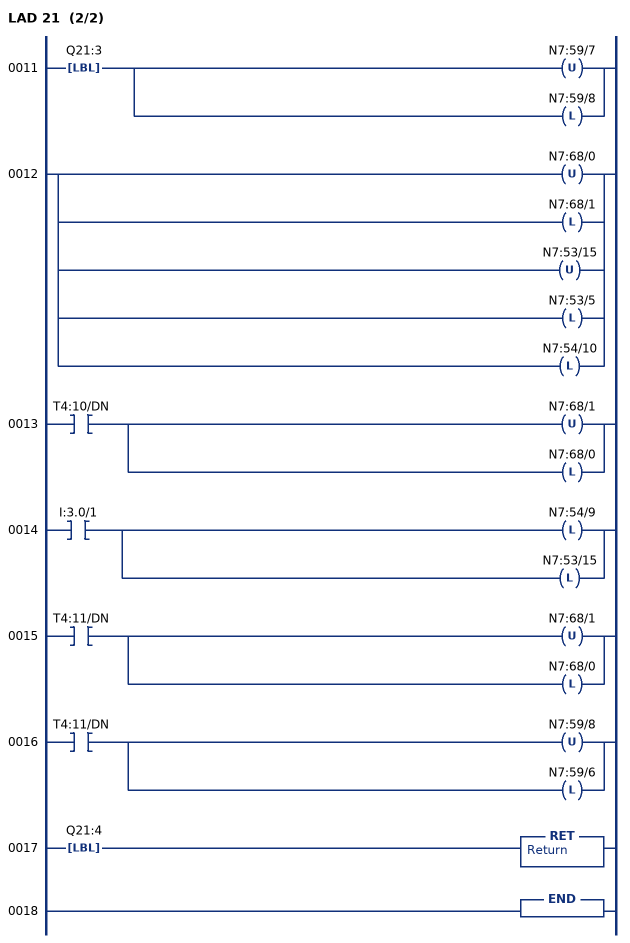
% Rung: 11 %
SOR LBL Q21:3 BST OTU N7:59/7 NXB OTL N7:59/8 BND EOR
% Rung: 12 %
SOR BST OTU N7:68/0 NXB OTL N7:68/1 NXB OTU N7:53/15 NXB OTL N7:53/5 NXB OTL N7:54/10 BND EOR
% Rung: 13 %
SOR XIC T4:10/DN BST OTU N7:68/1 NXB OTL N7:68/0 BND EOR
% Rung: 14 %
SOR XIC I:3.0/1 BST OTL N7:54/9 NXB OTL N7:53/15 BND EOR
% Rung: 15 %
SOR XIC T4:11/DN BST OTU N7:68/1 NXB OTL N7:68/0 BND EOR
% Rung: 16 %
SOR XIC T4:11/DN BST OTU N7:59/8 NXB OTL N7:59/6 BND EOR
% Rung: 17 %
SOR LBL Q21:4 RET EOR
% Rung: 18 %
SOR END EOR

LADDER 22
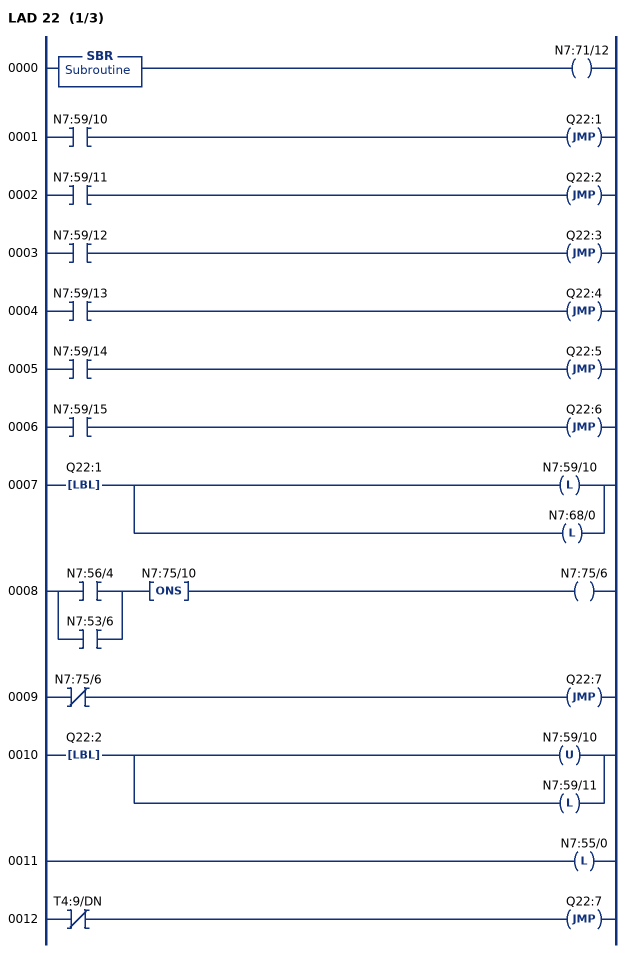
% Rung: 0 %
SOR SBR OTE N7:71/12 EOR
% Rung: 1 %
SOR XIC N7:59/10 JMP Q22:1 EOR
% Rung: 2 %
SOR XIC N7:59/11 JMP Q22:2 EOR
% Rung: 3 %
SOR XIC N7:59/12 JMP Q22:3 EOR
% Rung: 4 %
SOR XIC N7:59/13 JMP Q22:4 EOR
% Rung: 5 %
SOR XIC N7:59/14 JMP Q22:5 EOR
% Rung: 6 %
SOR XIC N7:59/15 JMP Q22:6 EOR
% Rung: 7 %
SOR LBL Q22:1 BST OTL N7:59/10 NXB OTL N7:68/0 BND EOR
% Rung: 8 %
SOR BST XIC N7:56/4 NXB XIC N7:53/6 BND OSR N7:75/10 OTE N7:75/6 EOR
% Rung: 9 %
SOR XIO N7:75/6 JMP Q22:7 EOR
% Rung: 10 %
SOR LBL Q22:2 BST OTU N7:59/10 NXB OTL N7:59/11 BND EOR
% Rung: 11 %
SOR OTL N7:55/0 EOR
% Rung: 12 %
SOR XIO T4:9/DN JMP Q22:7 EOR

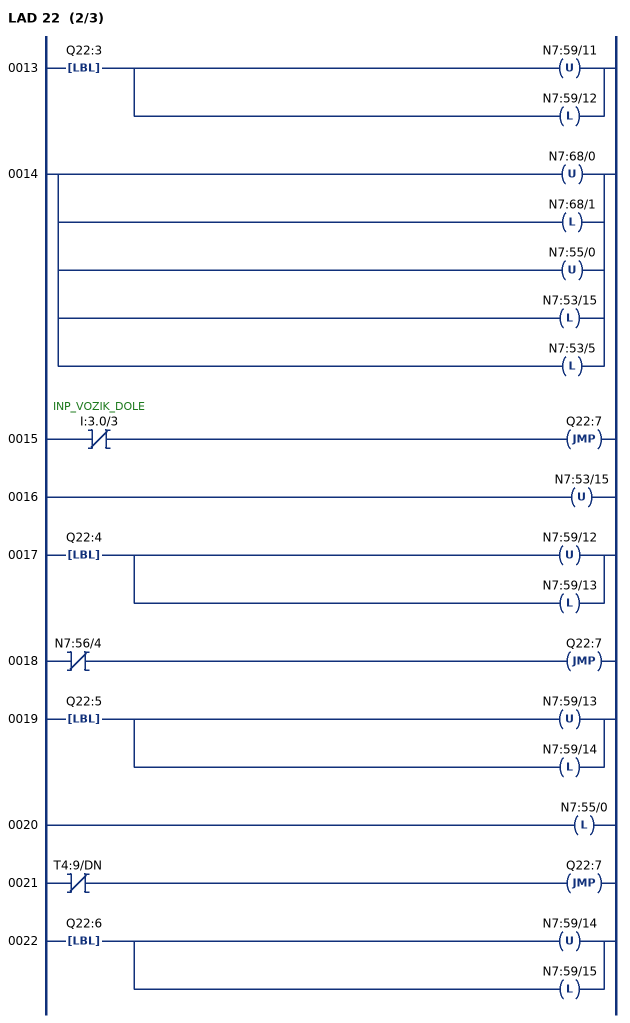
% Rung: 13 %
SOR LBL Q22:3 BST OTU N7:59/11 NXB OTL N7:59/12 BND EOR
% Rung: 14 %
SOR BST OTU N7:68/0 NXB OTL N7:68/1 NXB OTU N7:55/0 NXB OTL N7:53/15 NXB OTL N7:53/5 BND EOR
% Rung: 15 %
SOR XIO I:3.0/3 JMP Q22:7 EOR
%   I:3.0/3  INP_VOZIK_DOLE %
% Rung: 16 %
SOR OTU N7:53/15 EOR
% Rung: 17 %
SOR LBL Q22:4 BST OTU N7:59/12 NXB OTL N7:59/13 BND EOR
% Rung: 18 %
SOR XIO N7:56/4 JMP Q22:7 EOR
% Rung: 19 %
SOR LBL Q22:5 BST OTU N7:59/13 NXB OTL N7:59/14 BND EOR
% Rung: 20 %
SOR OTL N7:55/0 EOR
% Rung: 21 %
SOR XIO T4:9/DN JMP Q22:7 EOR
% Rung: 22 %
SOR LBL Q22:6 BST OTU N7:59/14 NXB OTL N7:59/15 BND EOR

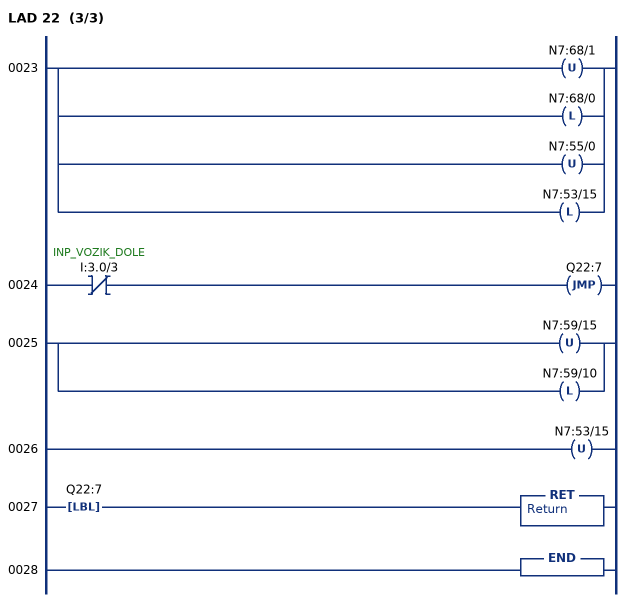
% Rung: 23 %
SOR BST OTU N7:68/1 NXB OTL N7:68/0 NXB OTU N7:55/0 NXB OTL N7:53/15 BND EOR
% Rung: 24 %
SOR XIO I:3.0/3 JMP Q22:7 EOR
%   I:3.0/3  INP_VOZIK_DOLE %
% Rung: 25 %
SOR BST OTU N7:59/15 NXB OTL N7:59/10 BND EOR
% Rung: 26 %
SOR OTU N7:53/15 EOR
% Rung: 27 %
SOR LBL Q22:7 RET EOR
% Rung: 28 %
SOR END EOR

LADDER 23
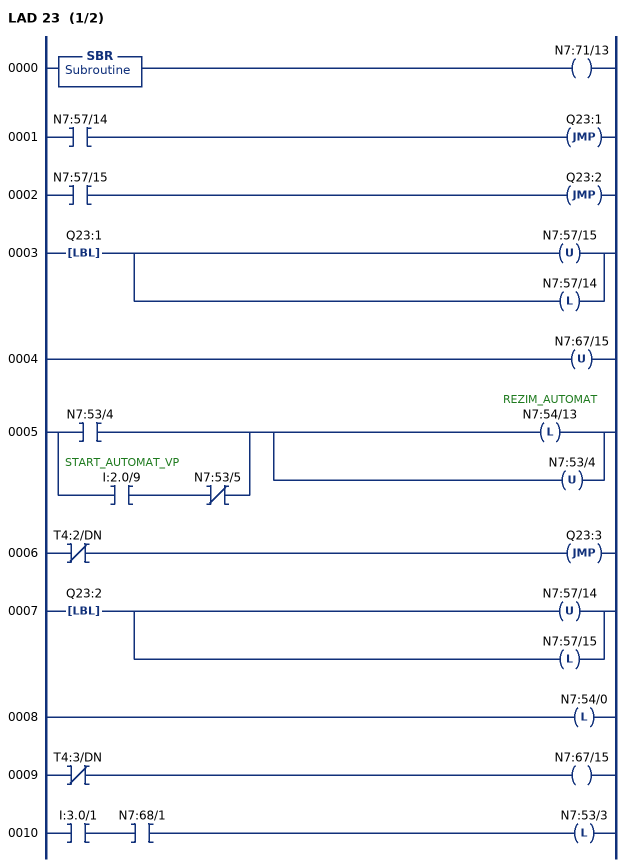
% Rung: 0 %
SOR SBR OTE N7:71/13 EOR
% Rung: 1 %
SOR XIC N7:57/14 JMP Q23:1 EOR
% Rung: 2 %
SOR XIC N7:57/15 JMP Q23:2 EOR
% Rung: 3 %
SOR LBL Q23:1 BST OTU N7:57/15 NXB OTL N7:57/14 BND EOR
% Rung: 4 %
SOR OTU N7:67/15 EOR
% Rung: 5 %
SOR BST XIC N7:53/4 NXB XIC I:2.0/9 XIO N7:53/5 BND BST OTL N7:54/13 NXB OTU N7:53/4 BND EOR
%   I:2.0/9  START_AUTOMAT_VP %
%   N7:54/13  REZIM_AUTOMAT %
% Rung: 6 %
SOR XIO T4:2/DN JMP Q23:3 EOR
% Rung: 7 %
SOR LBL Q23:2 BST OTU N7:57/14 NXB OTL N7:57/15 BND EOR
% Rung: 8 %
SOR OTL N7:54/0 EOR
% Rung: 9 %
SOR XIO T4:3/DN OTE N7:67/15 EOR
% Rung: 10 %
SOR XIC I:3.0/1 XIC N7:68/1 OTL N7:53/3 EOR

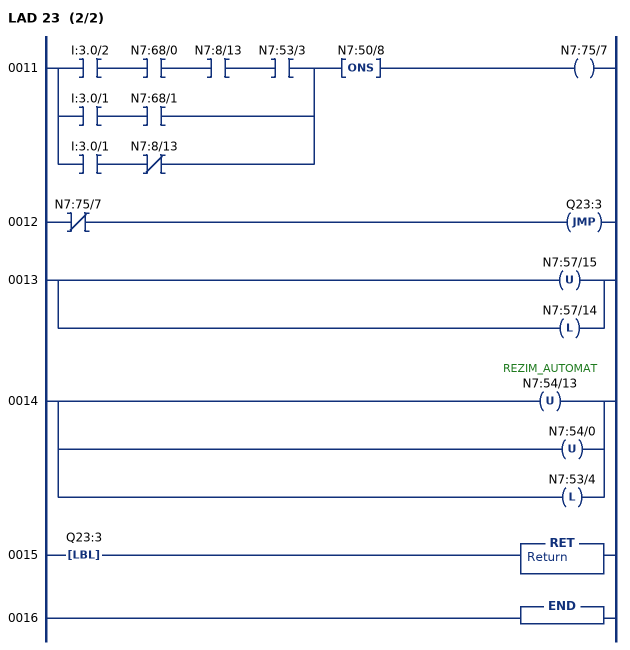
% Rung: 11 %
SOR BST XIC I:3.0/2 XIC N7:68/0 XIC N7:8/13 XIC N7:53/3 NXB XIC I:3.0/1 XIC N7:68/1 NXB XIC I:3.0/1 XIO N7:8/13 BND OSR N7:50/8 OTE N7:75/7 EOR
% Rung: 12 %
SOR XIO N7:75/7 JMP Q23:3 EOR
% Rung: 13 %
SOR BST OTU N7:57/15 NXB OTL N7:57/14 BND EOR
% Rung: 14 %
SOR BST OTU N7:54/13 NXB OTU N7:54/0 NXB OTL N7:53/4 BND EOR
%   N7:54/13  REZIM_AUTOMAT %
% Rung: 15 %
SOR LBL Q23:3 RET EOR
% Rung: 16 %
SOR END EOR

LADDER 24
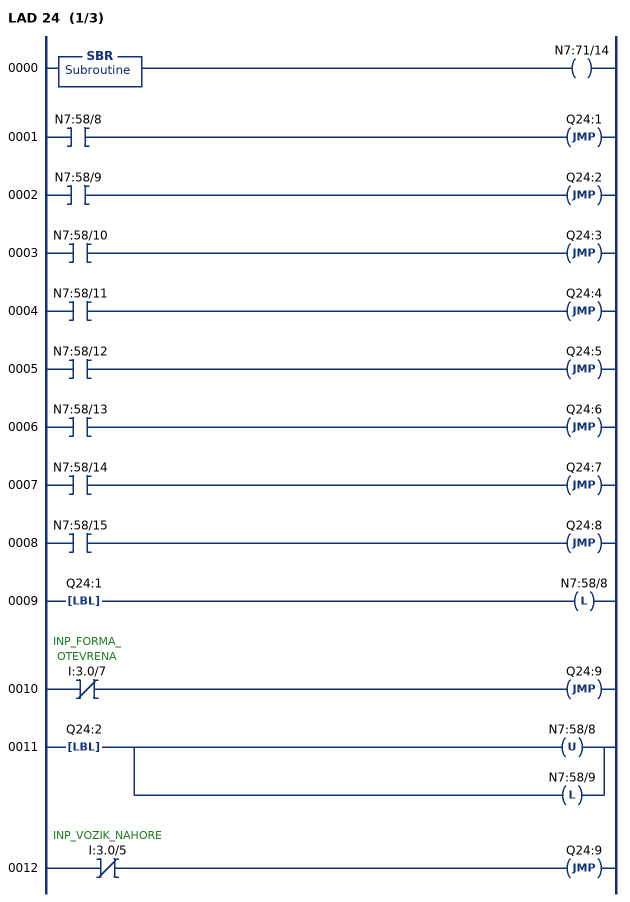
% Rung: 0 %
SOR SBR OTE N7:71/14 EOR
% Rung: 1 %
SOR XIC N7:58/8 JMP Q24:1 EOR
% Rung: 2 %
SOR XIC N7:58/9 JMP Q24:2 EOR
% Rung: 3 %
SOR XIC N7:58/10 JMP Q24:3 EOR
% Rung: 4 %
SOR XIC N7:58/11 JMP Q24:4 EOR
% Rung: 5 %
SOR XIC N7:58/12 JMP Q24:5 EOR
% Rung: 6 %
SOR XIC N7:58/13 JMP Q24:6 EOR
% Rung: 7 %
SOR XIC N7:58/14 JMP Q24:7 EOR
% Rung: 8 %
SOR XIC N7:58/15 JMP Q24:8 EOR
% Rung: 9 %
SOR LBL Q24:1 OTL N7:58/8 EOR
% Rung: 10 %
SOR XIO I:3.0/7 JMP Q24:9 EOR
%   I:3.0/7  INP_FORMA_OTEVRENA %
% Rung: 11 %
SOR LBL Q24:2 BST OTU N7:58/8 NXB OTL N7:58/9 BND EOR
% Rung: 12 %
SOR XIO I:3.0/5 JMP Q24:9 EOR
%   I:3.0/5  INP_VOZIK_NAHORE %

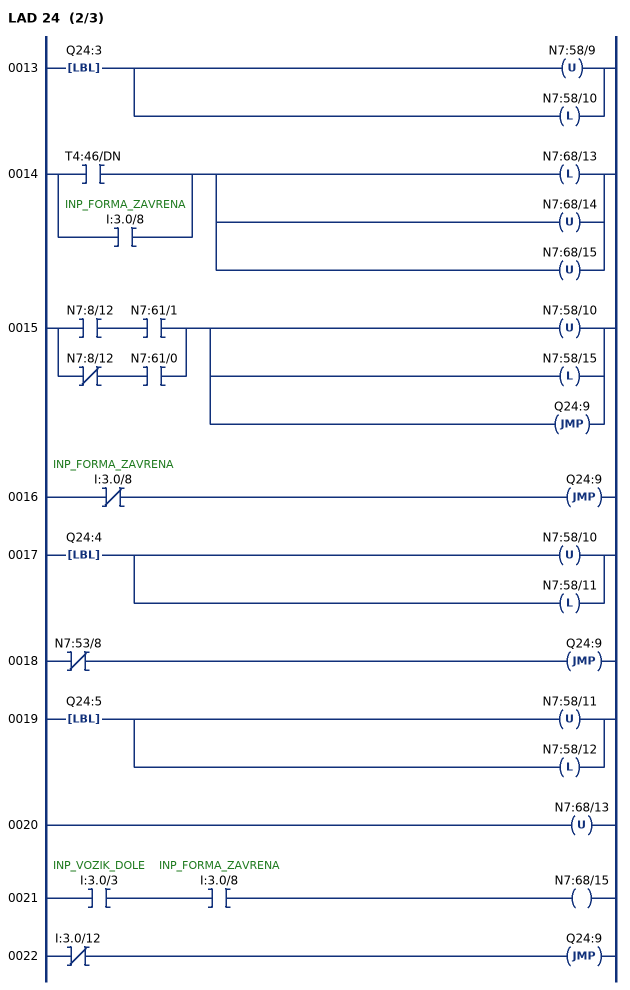
% Rung: 13 %
SOR LBL Q24:3 BST OTU N7:58/9 NXB OTL N7:58/10 BND EOR
% Rung: 14 %
SOR BST XIC T4:46/DN NXB XIC I:3.0/8 BND BST OTL N7:68/13 NXB BST OTU N7:68/14 NXB OTU N7:68/15 BND BND EOR
%   I:3.0/8  INP_FORMA_ZAVRENA %
% Rung: 15 %
SOR BST XIC N7:8/12 XIC N7:61/1 NXB XIO N7:8/12 XIC N7:61/0 BND BST OTU N7:58/10 NXB OTL N7:58/15 NXB JMP Q24:9 BND EOR
% Rung: 16 %
SOR XIO I:3.0/8 JMP Q24:9 EOR
%   I:3.0/8  INP_FORMA_ZAVRENA %
% Rung: 17 %
SOR LBL Q24:4 BST OTU N7:58/10 NXB OTL N7:58/11 BND EOR
% Rung: 18 %
SOR XIO N7:53/8 JMP Q24:9 EOR
% Rung: 19 %
SOR LBL Q24:5 BST OTU N7:58/11 NXB OTL N7:58/12 BND EOR
% Rung: 20 %
SOR OTU N7:68/13 EOR
% Rung: 21 %
SOR XIC I:3.0/3 XIC I:3.0/8 OTE N7:68/15 EOR
%   I:3.0/3  INP_VOZIK_DOLE %
%   I:3.0/8  INP_FORMA_ZAVRENA %
% Rung: 22 %
SOR XIO I:3.0/12 JMP Q24:9 EOR

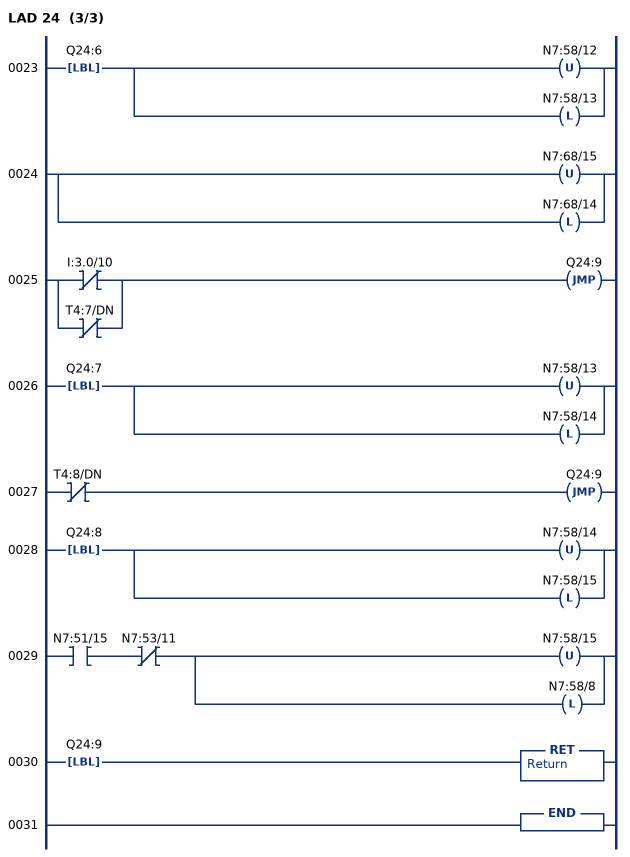
% Rung: 23 %
SOR LBL Q24:6 BST OTU N7:58/12 NXB OTL N7:58/13 BND EOR
% Rung: 24 %
SOR BST OTU N7:68/15 NXB OTL N7:68/14 BND EOR
% Rung: 25 %
SOR BST XIO I:3.0/10 NXB XIO T4:7/DN BND JMP Q24:9 EOR
% Rung: 26 %
SOR LBL Q24:7 BST OTU N7:58/13 NXB OTL N7:58/14 BND EOR
% Rung: 27 %
SOR XIO T4:8/DN JMP Q24:9 EOR
% Rung: 28 %
SOR LBL Q24:8 BST OTU N7:58/14 NXB OTL N7:58/15 BND EOR
% Rung: 29 %
SOR XIC N7:51/15 XIO N7:53/11 BST OTU N7:58/15 NXB OTL N7:58/8 BND EOR
% Rung: 30 %
SOR LBL Q24:9 RET EOR
% Rung: 31 %
SOR END EOR

LADDER 25
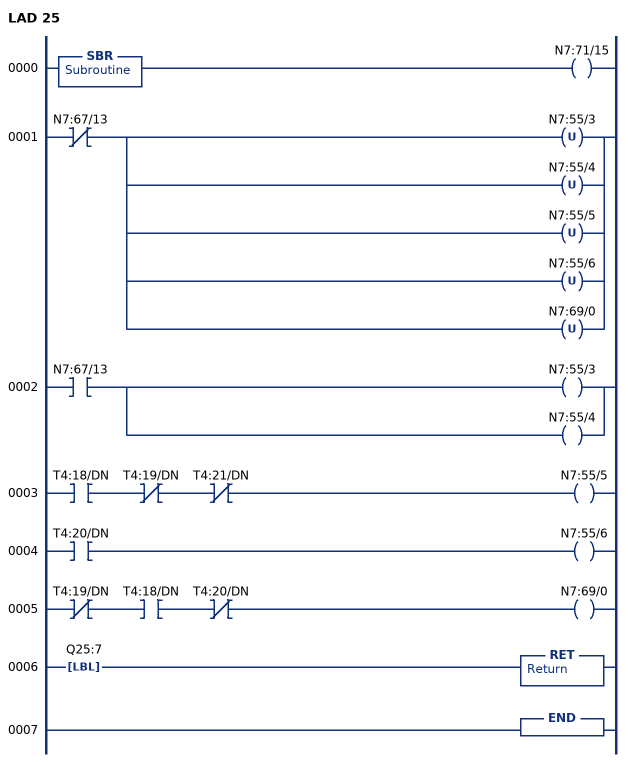
% Rung: 0 %
SOR SBR OTE N7:71/15 EOR
% Rung: 1 %
SOR XIO N7:67/13 BST OTU N7:55/3 NXB OTU N7:55/4 NXB OTU N7:55/5 NXB OTU N7:55/6 NXB OTU N7:69/0 BND EOR
% Rung: 2 %
SOR XIC N7:67/13 BST OTE N7:55/3 NXB OTE N7:55/4 BND EOR
% Rung: 3 %
SOR XIC T4:18/DN XIO T4:19/DN XIO T4:21/DN OTE N7:55/5 EOR
% Rung: 4 %
SOR XIC T4:20/DN OTE N7:55/6 EOR
% Rung: 5 %
SOR XIO T4:19/DN XIC T4:18/DN XIO T4:20/DN OTE N7:69/0 EOR
% Rung: 6 %
SOR LBL Q25:7 RET EOR
% Rung: 7 %
SOR END EOR

LADDER 26
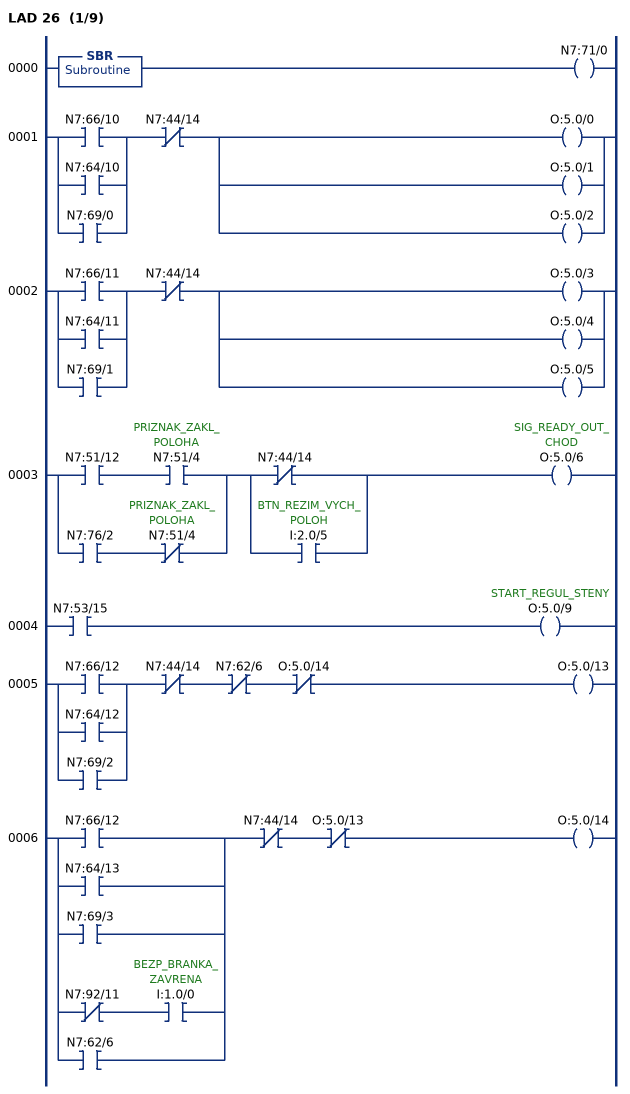
% Rung: 0 %
SOR SBR OTE N7:71/0 EOR
% Rung: 1 %
SOR BST XIC N7:66/10 NXB XIC N7:64/10 NXB XIC N7:69/0 BND XIO N7:44/14 BST OTE O:5.0/0 NXB OTE O:5.0/1 NXB OTE O:5.0/2 BND EOR
% Rung: 2 %
SOR BST XIC N7:66/11 NXB XIC N7:64/11 NXB XIC N7:69/1 BND XIO N7:44/14 BST OTE O:5.0/3 NXB OTE O:5.0/4 NXB OTE O:5.0/5 BND EOR
% Rung: 3 %
SOR BST XIC N7:51/12 XIC N7:51/4 NXB XIC N7:76/2 XIO N7:51/4 BND BST XIO N7:44/14 NXB XIC I:2.0/5 BND OTE O:5.0/6 EOR
%   N7:51/4  PRIZNAK_ZAKL_POLOHA %
%   I:2.0/5  BTN_REZIM_VYCH_POLOH %
%   O:5.0/6  SIG_READY_OUT_CHOD %
% Rung: 4 %
SOR XIC N7:53/15 OTE O:5.0/9 EOR
%   O:5.0/9  START_REGUL_STENY %
% Rung: 5 %
SOR BST XIC N7:66/12 NXB XIC N7:64/12 NXB XIC N7:69/2 BND XIO N7:44/14 XIO N7:62/6 XIO O:5.0/14 OTE O:5.0/13 EOR
% Rung: 6 %
SOR BST XIC N7:66/12 NXB XIC N7:64/13 NXB XIC N7:69/3 NXB BST XIO N7:92/11 XIC I:1.0/0 NXB XIC N7:62/6 BND BND XIO N7:44/14 XIO O:5.0/13 OTE O:5.0/14 EOR
%   I:1.0/0  BEZP_BRANKA_ZAVRENA %

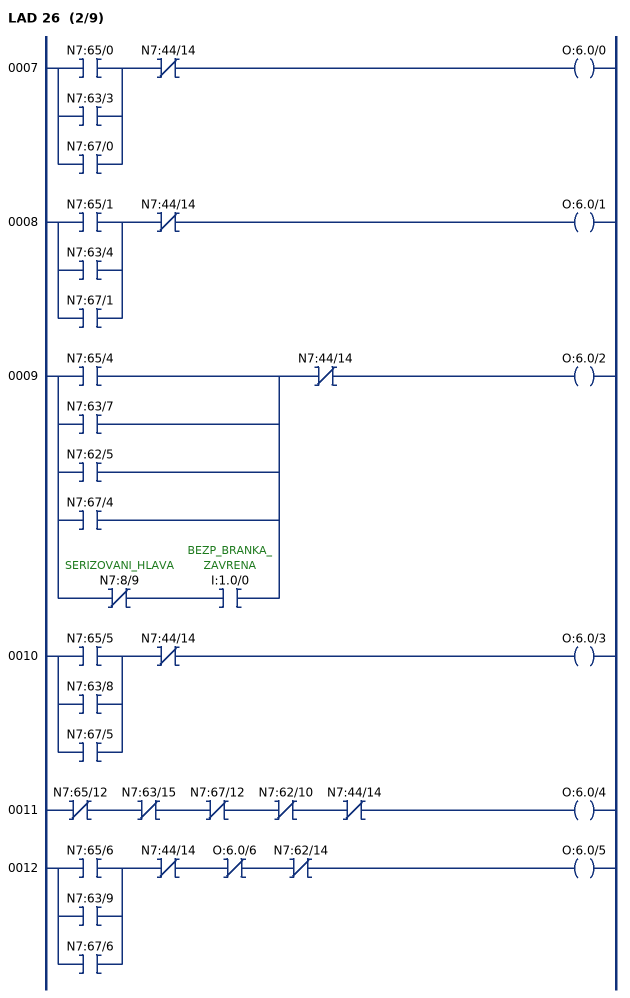
% Rung: 7 %
SOR BST XIC N7:65/0 NXB XIC N7:63/3 NXB XIC N7:67/0 BND XIO N7:44/14 OTE O:6.0/0 EOR
% Rung: 8 %
SOR BST XIC N7:65/1 NXB XIC N7:63/4 NXB XIC N7:67/1 BND XIO N7:44/14 OTE O:6.0/1 EOR
% Rung: 9 %
SOR BST XIC N7:65/4 NXB XIC N7:63/7 NXB XIC N7:62/5 NXB XIC N7:67/4 NXB XIO N7:8/9 XIC I:1.0/0 BND XIO N7:44/14 OTE O:6.0/2 EOR
%   N7:8/9  SERIZOVANI_HLAVA %
%   I:1.0/0  BEZP_BRANKA_ZAVRENA %
% Rung: 10 %
SOR BST XIC N7:65/5 NXB XIC N7:63/8 NXB XIC N7:67/5 BND XIO N7:44/14 OTE O:6.0/3 EOR
% Rung: 11 %
SOR XIO N7:65/12 XIO N7:63/15 XIO N7:67/12 XIO N7:62/10 XIO N7:44/14 OTE O:6.0/4 EOR
% Rung: 12 %
SOR BST XIC N7:65/6 NXB XIC N7:63/9 NXB XIC N7:67/6 BND XIO N7:44/14 XIO O:6.0/6 XIO N7:62/14 OTE O:6.0/5 EOR

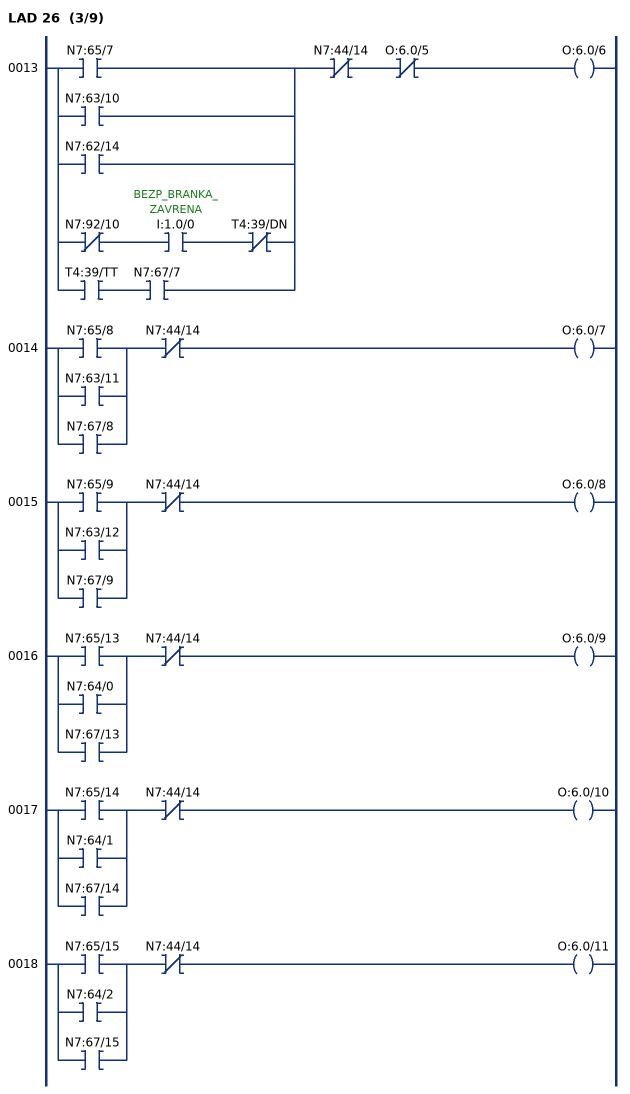
% Rung: 13 %
SOR BST XIC N7:65/7 NXB BST XIC N7:63/10 NXB XIC N7:62/14 BND NXB XIO N7:92/10 XIC I:1.0/0 XIO T4:39/DN NXB XIC T4:39/TT XIC N7:67/7 BND XIO N7:44/14 XIO O:6.0/5 OTE O:6.0/6 EOR
%   I:1.0/0  BEZP_BRANKA_ZAVRENA %
% Rung: 14 %
SOR BST XIC N7:65/8 NXB XIC N7:63/11 NXB XIC N7:67/8 BND XIO N7:44/14 OTE O:6.0/7 EOR
% Rung: 15 %
SOR BST XIC N7:65/9 NXB XIC N7:63/12 NXB XIC N7:67/9 BND XIO N7:44/14 OTE O:6.0/8 EOR
% Rung: 16 %
SOR BST XIC N7:65/13 NXB XIC N7:64/0 NXB XIC N7:67/13 BND XIO N7:44/14 OTE O:6.0/9 EOR
% Rung: 17 %
SOR BST XIC N7:65/14 NXB XIC N7:64/1 NXB XIC N7:67/14 BND XIO N7:44/14 OTE O:6.0/10 EOR
% Rung: 18 %
SOR BST XIC N7:65/15 NXB XIC N7:64/2 NXB XIC N7:67/15 BND XIO N7:44/14 OTE O:6.0/11 EOR

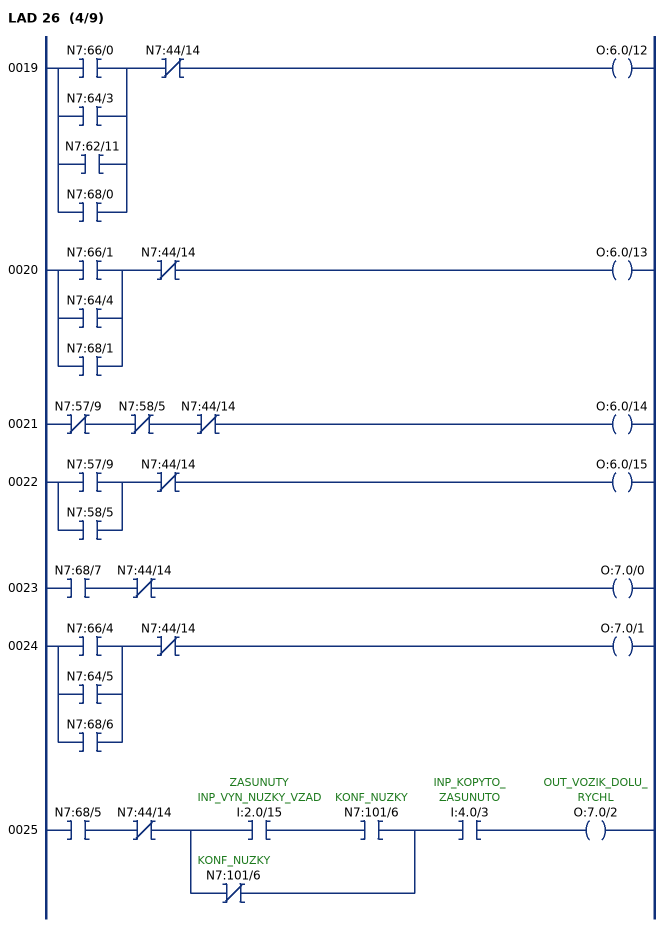
% Rung: 19 %
SOR BST XIC N7:66/0 NXB XIC N7:64/3 NXB XIC N7:62/11 NXB XIC N7:68/0 BND XIO N7:44/14 OTE O:6.0/12 EOR
% Rung: 20 %
SOR BST XIC N7:66/1 NXB XIC N7:64/4 NXB XIC N7:68/1 BND XIO N7:44/14 OTE O:6.0/13 EOR
% Rung: 21 %
SOR XIO N7:57/9 XIO N7:58/5 XIO N7:44/14 OTE O:6.0/14 EOR
% Rung: 22 %
SOR BST XIC N7:57/9 NXB XIC N7:58/5 BND XIO N7:44/14 OTE O:6.0/15 EOR
% Rung: 23 %
SOR XIC N7:68/7 XIO N7:44/14 OTE O:7.0/0 EOR
% Rung: 24 %
SOR BST XIC N7:66/4 NXB XIC N7:64/5 NXB XIC N7:68/6 BND XIO N7:44/14 OTE O:7.0/1 EOR
% Rung: 25 %
SOR XIC N7:68/5 XIO N7:44/14 BST XIC I:2.0/15 XIC N7:101/6 NXB XIO N7:101/6 BND XIC I:4.0/3 OTE O:7.0/2 EOR
%   I:2.0/15  INP_VYN_NUZKY_VZAD  "ZASUNUTY" %
%   N7:101/6  KONF_NUZKY %
%   I:4.0/3  INP_KOPYTO_ZASUNUTO %
%   O:7.0/2  OUT_VOZIK_DOLU_RYCHL %

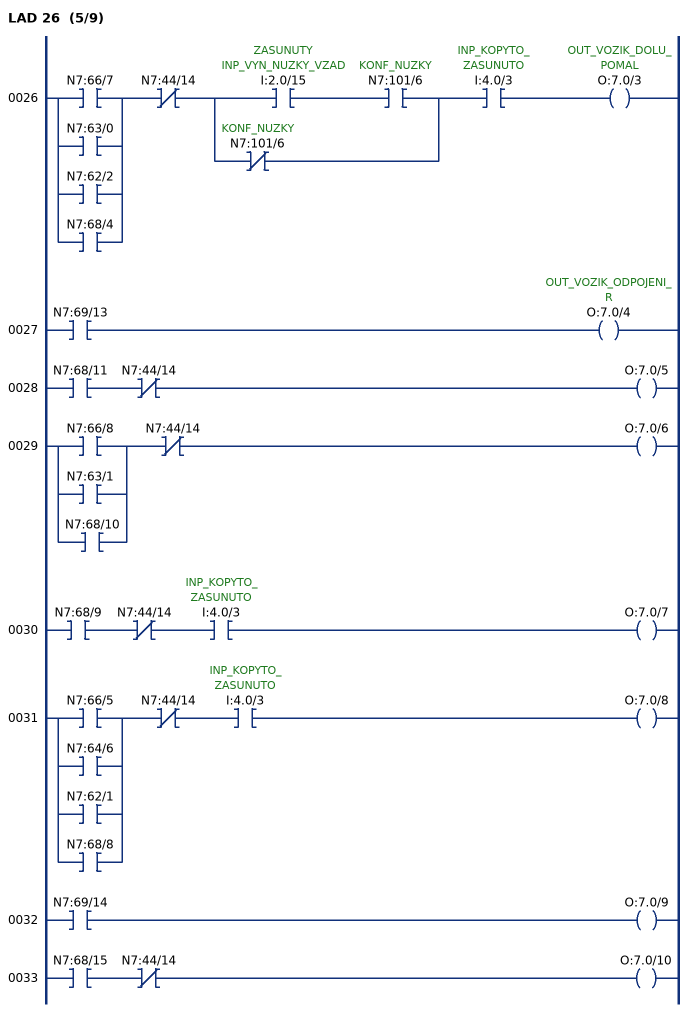
% Rung: 26 %
SOR BST XIC N7:66/7 NXB XIC N7:63/0 NXB XIC N7:62/2 NXB XIC N7:68/4 BND XIO N7:44/14 BST XIC I:2.0/15 XIC N7:101/6 NXB XIO N7:101/6 BND XIC I:4.0/3 OTE O:7.0/3 EOR
%   I:2.0/15  INP_VYN_NUZKY_VZAD  "ZASUNUTY" %
%   N7:101/6  KONF_NUZKY %
%   I:4.0/3  INP_KOPYTO_ZASUNUTO %
%   O:7.0/3  OUT_VOZIK_DOLU_POMAL %
% Rung: 27 %
SOR XIC N7:69/13 OTE O:7.0/4 EOR
%   O:7.0/4  OUT_VOZIK_ODPOJENI_R %
% Rung: 28 %
SOR XIC N7:68/11 XIO N7:44/14 OTE O:7.0/5 EOR
% Rung: 29 %
SOR BST XIC N7:66/8 NXB XIC N7:63/1 NXB XIC N7:68/10 BND XIO N7:44/14 OTE O:7.0/6 EOR
% Rung: 30 %
SOR XIC N7:68/9 XIO N7:44/14 XIC I:4.0/3 OTE O:7.0/7 EOR
%   I:4.0/3  INP_KOPYTO_ZASUNUTO %
% Rung: 31 %
SOR BST XIC N7:66/5 NXB XIC N7:64/6 NXB XIC N7:62/1 NXB XIC N7:68/8 BND XIO N7:44/14 XIC I:4.0/3 OTE O:7.0/8 EOR
%   I:4.0/3  INP_KOPYTO_ZASUNUTO %
% Rung: 32 %
SOR XIC N7:69/14 OTE O:7.0/9 EOR
% Rung: 33 %
SOR XIC N7:68/15 XIO N7:44/14 OTE O:7.0/10 EOR

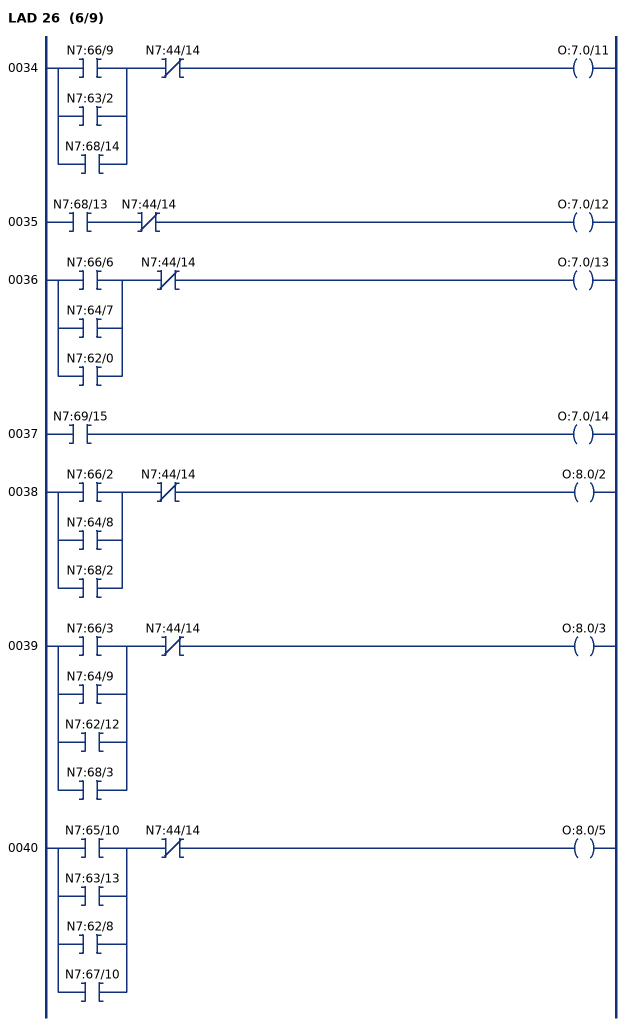
% Rung: 34 %
SOR BST XIC N7:66/9 NXB XIC N7:63/2 NXB XIC N7:68/14 BND XIO N7:44/14 OTE O:7.0/11 EOR
% Rung: 35 %
SOR XIC N7:68/13 XIO N7:44/14 OTE O:7.0/12 EOR
% Rung: 36 %
SOR BST XIC N7:66/6 NXB XIC N7:64/7 NXB XIC N7:62/0 BND XIO N7:44/14 OTE O:7.0/13 EOR
% Rung: 37 %
SOR XIC N7:69/15 OTE O:7.0/14 EOR
% Rung: 38 %
SOR BST XIC N7:66/2 NXB XIC N7:64/8 NXB XIC N7:68/2 BND XIO N7:44/14 OTE O:8.0/2 EOR
% Rung: 39 %
SOR BST XIC N7:66/3 NXB XIC N7:64/9 NXB XIC N7:62/12 NXB XIC N7:68/3 BND XIO N7:44/14 OTE O:8.0/3 EOR
% Rung: 40 %
SOR BST XIC N7:65/10 NXB XIC N7:63/13 NXB XIC N7:62/8 NXB XIC N7:67/10 BND XIO N7:44/14 OTE O:8.0/5 EOR

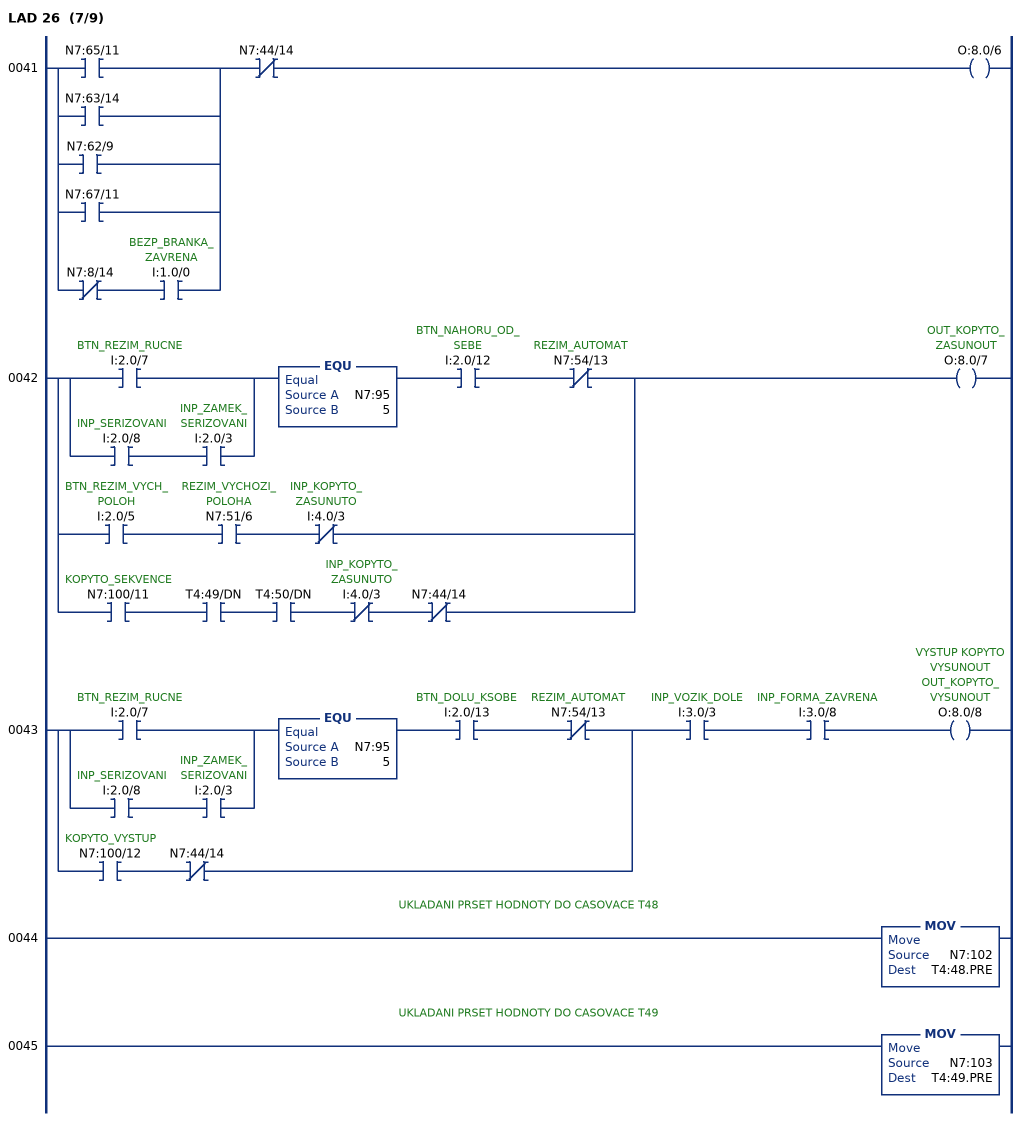
% Rung: 41 %
SOR BST XIC N7:65/11 NXB XIC N7:63/14 NXB XIC N7:62/9 NXB XIC N7:67/11 NXB XIO N7:8/14 XIC I:1.0/0 BND XIO N7:44/14 OTE O:8.0/6 EOR
%   I:1.0/0  BEZP_BRANKA_ZAVRENA %
% Rung: 42 %
SOR BST BST XIC I:2.0/7 NXB XIC I:2.0/8 XIC I:2.0/3 BND EQU N7:95 5 XIC I:2.0/12 XIO N7:54/13 NXB XIC I:2.0/5 XIC N7:51/6 XIO I:4.0/3 NXB XIC N7:100/11 XIC T4:49/DN XIC T4:50/DN XIO I:4.0/3 XIO N7:44/14 BND OTE O:8.0/7 EOR
%   I:2.0/7  BTN_REZIM_RUCNE %
%   I:2.0/8  INP_SERIZOVANI %
%   I:2.0/3  INP_ZAMEK_SERIZOVANI %
%   I:2.0/12  BTN_NAHORU_OD_SEBE %
%   N7:54/13  REZIM_AUTOMAT %
%   I:2.0/5  BTN_REZIM_VYCH_POLOH %
%   N7:51/6  REZIM_VYCHOZI_POLOHA %
%   I:4.0/3  INP_KOPYTO_ZASUNUTO %
%   N7:100/11  KOPYTO_SEKVENCE %
%   O:8.0/7  OUT_KOPYTO_ZASUNOUT %
% Rung: 43 %
SOR BST BST XIC I:2.0/7 NXB XIC I:2.0/8 XIC I:2.0/3 BND EQU N7:95 5 XIC I:2.0/13 XIO N7:54/13 NXB XIC N7:100/12 XIO N7:44/14 BND XIC I:3.0/3 XIC I:3.0/8 OTE O:8.0/8 EOR
%   I:2.0/7  BTN_REZIM_RUCNE %
%   I:2.0/8  INP_SERIZOVANI %
%   I:2.0/3  INP_ZAMEK_SERIZOVANI %
%   I:2.0/13  BTN_DOLU_KSOBE %
%   N7:54/13  REZIM_AUTOMAT %
%   N7:100/12  KOPYTO_VYSTUP %
%   I:3.0/3  INP_VOZIK_DOLE %
%   I:3.0/8  INP_FORMA_ZAVRENA %
%   O:8.0/8  OUT_KOPYTO_VYSUNOUT  "VYSTUP KOPYTO VYSUNOUT" %
% Rung: 44 %
% UKLADANI PRSET HODNOTY DO CASOVACE T48 %
SOR MOV N7:102 T4:48.PRE EOR
%   N7:102  CASOVAC_T48_PRESET %
% Rung: 45 %
% UKLADANI PRSET HODNOTY DO CASOVACE T49 %
SOR MOV N7:103 T4:49.PRE EOR
%   N7:103  CASOVAC_T49_PRESET %

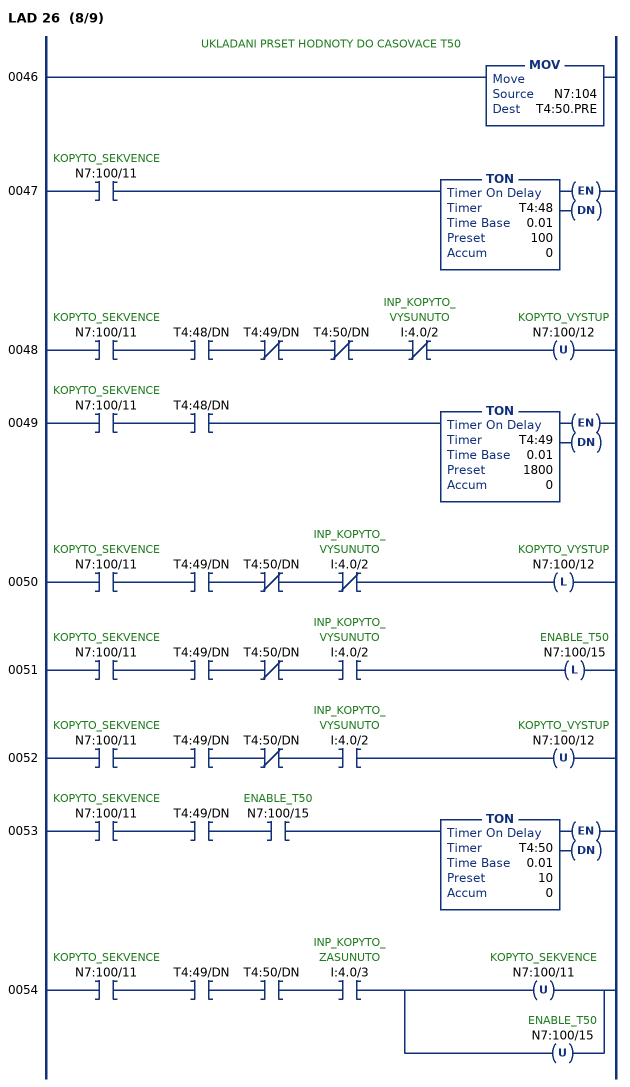
% Rung: 46 %
% UKLADANI PRSET HODNOTY DO CASOVACE T50 %
SOR MOV N7:104 T4:50.PRE EOR
%   N7:104  CASOVAC_T50_PRESET %
% Rung: 47 %
SOR XIC N7:100/11 TON T4:48 0.01 100 0 EOR
%   N7:100/11  KOPYTO_SEKVENCE %
% Rung: 48 %
SOR XIC N7:100/11 XIC T4:48/DN XIO T4:49/DN XIO T4:50/DN XIO I:4.0/2 OTU N7:100/12 EOR
%   N7:100/11  KOPYTO_SEKVENCE %
%   I:4.0/2  INP_KOPYTO_VYSUNUTO %
%   N7:100/12  KOPYTO_VYSTUP %
% Rung: 49 %
SOR XIC N7:100/11 XIC T4:48/DN TON T4:49 0.01 1800 0 EOR
%   N7:100/11  KOPYTO_SEKVENCE %
% Rung: 50 %
SOR XIC N7:100/11 XIC T4:49/DN XIO T4:50/DN XIO I:4.0/2 OTL N7:100/12 EOR
%   N7:100/11  KOPYTO_SEKVENCE %
%   I:4.0/2  INP_KOPYTO_VYSUNUTO %
%   N7:100/12  KOPYTO_VYSTUP %
% Rung: 51 %
SOR XIC N7:100/11 XIC T4:49/DN XIO T4:50/DN XIC I:4.0/2 OTL N7:100/15 EOR
%   N7:100/11  KOPYTO_SEKVENCE %
%   I:4.0/2  INP_KOPYTO_VYSUNUTO %
%   N7:100/15  ENABLE_T50 %
% Rung: 52 %
SOR XIC N7:100/11 XIC T4:49/DN XIO T4:50/DN XIC I:4.0/2 OTU N7:100/12 EOR
%   N7:100/11  KOPYTO_SEKVENCE %
%   I:4.0/2  INP_KOPYTO_VYSUNUTO %
%   N7:100/12  KOPYTO_VYSTUP %
% Rung: 53 %
SOR XIC N7:100/11 XIC T4:49/DN XIC N7:100/15 TON T4:50 0.01 10 0 EOR
%   N7:100/11  KOPYTO_SEKVENCE %
%   N7:100/15  ENABLE_T50 %
% Rung: 54 %
SOR XIC N7:100/11 XIC T4:49/DN XIC T4:50/DN XIC I:4.0/3 BST OTU N7:100/11 NXB OTU N7:100/15 BND EOR
%   N7:100/11  KOPYTO_SEKVENCE %
%   I:4.0/3  INP_KOPYTO_ZASUNUTO %
%   N7:100/15  ENABLE_T50 %

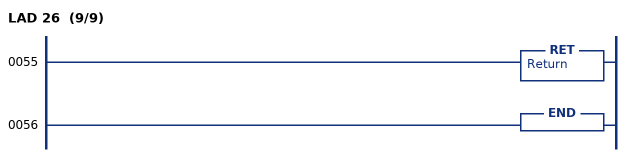
% Rung: 55 %
SOR RET EOR
% Rung: 56 %
SOR END EOR

LADDER 27
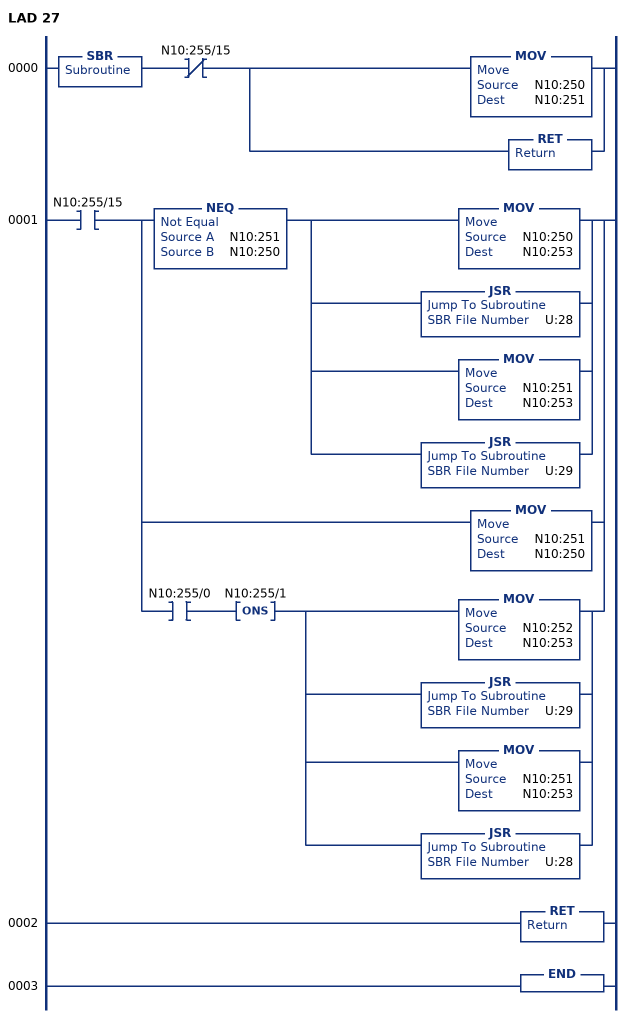
% Rung: 0 %
SOR SBR XIO N10:255/15 BST MOV N10:250 N10:251 NXB RET BND EOR
% Rung: 1 %
SOR XIC N10:255/15 BST NEQ N10:251 N10:250 BST MOV N10:250 N10:253 NXB JSR U:28 NXB MOV N10:251 N10:253 NXB JSR U:29 BND NXB MOV N10:251 N10:250 NXB XIC N10:255/0 OSR N10:255/1 BST MOV N10:252 N10:253 NXB JSR U:29 NXB MOV N10:251 N10:253 NXB JSR U:28 BND BND EOR
% Rung: 2 %
SOR RET EOR
% Rung: 3 %
SOR END EOR

LADDER 28
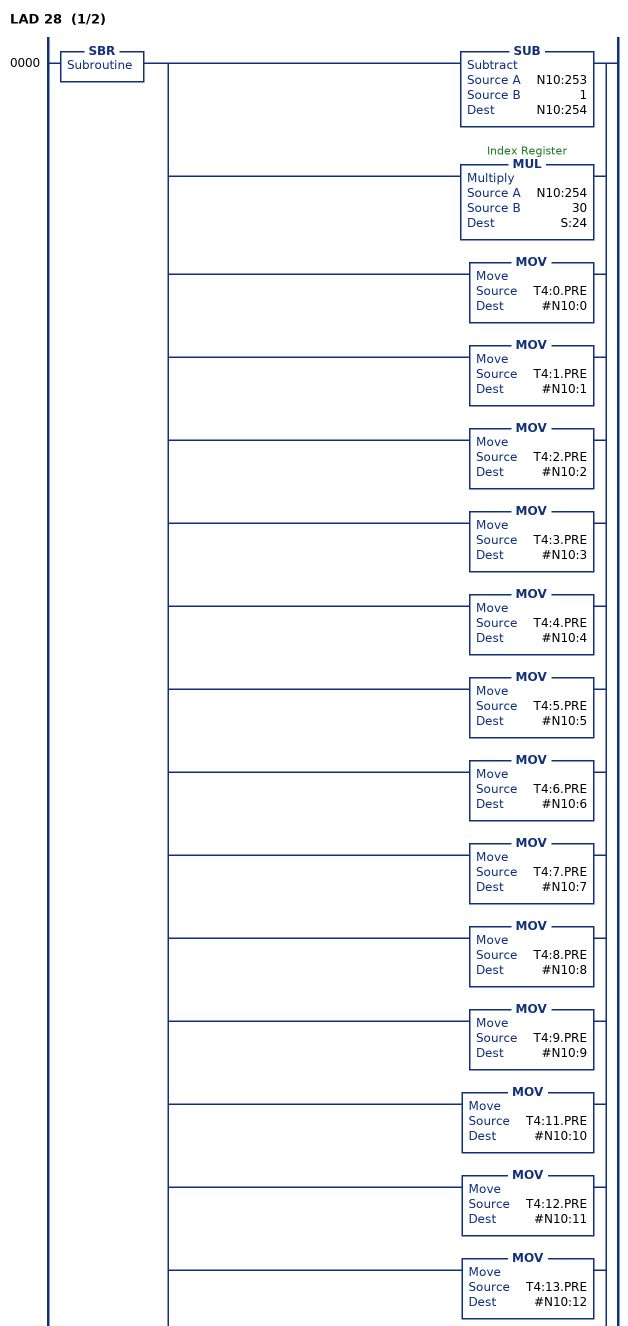
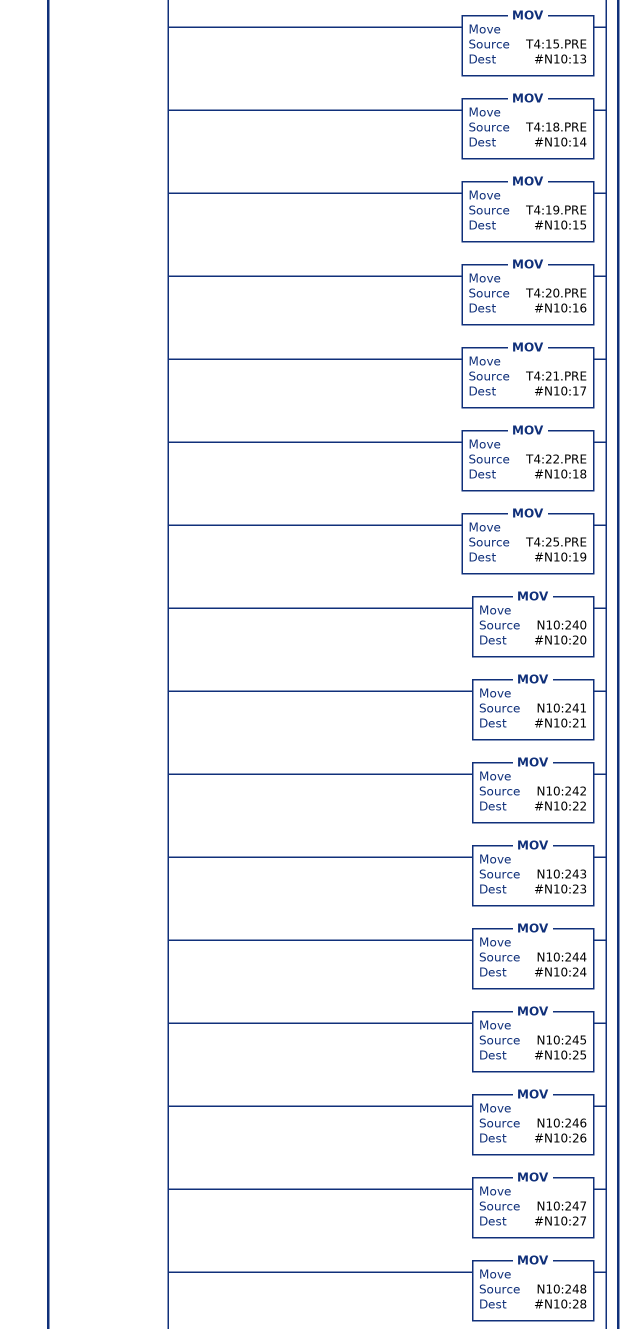
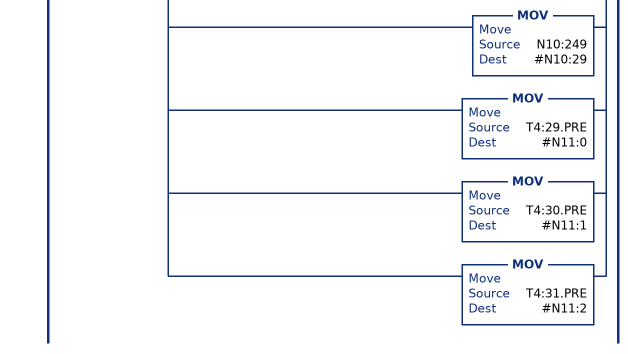
% Rung: 0 %
SOR SBR BST SUB N10:253 1 N10:254 NXB MUL N10:254 30 S:24 NXB MOV T4:0.PRE #N10:0 NXB MOV T4:1.PRE #N10:1 NXB MOV T4:2.PRE #N10:2 NXB MOV T4:3.PRE #N10:3 NXB MOV T4:4.PRE #N10:4 NXB MOV T4:5.PRE #N10:5 NXB MOV T4:6.PRE #N10:6 NXB MOV T4:7.PRE #N10:7 NXB MOV T4:8.PRE #N10:8 NXB MOV T4:9.PRE #N10:9 NXB MOV T4:11.PRE #N10:10 NXB MOV T4:12.PRE #N10:11 NXB MOV T4:13.PRE #N10:12 NXB MOV T4:15.PRE #N10:13 NXB MOV T4:18.PRE #N10:14 NXB MOV T4:19.PRE #N10:15 NXB MOV T4:20.PRE #N10:16 NXB MOV T4:21.PRE #N10:17 NXB MOV T4:22.PRE #N10:18 NXB MOV T4:25.PRE #N10:19 NXB MOV N10:240 #N10:20 NXB MOV N10:241 #N10:21 NXB MOV N10:242 #N10:22 NXB MOV N10:243 #N10:23 NXB MOV N10:244 #N10:24 NXB MOV N10:245 #N10:25 NXB MOV N10:246 #N10:26 NXB MOV N10:247 #N10:27 NXB MOV N10:248 #N10:28 NXB MOV N10:249 #N10:29 NXB MOV T4:29.PRE #N11:0 NXB MOV T4:30.PRE #N11:1 NXB MOV T4:31.PRE #N11:2 BND EOR
%   S:24  "Index Register" %

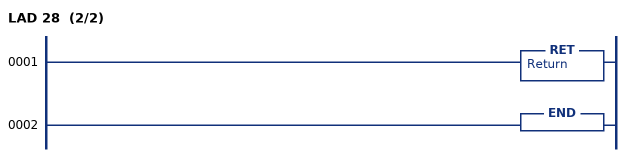
% Rung: 1 %
SOR RET EOR
% Rung: 2 %
SOR END EOR

LADDER 29
